FUNCTION_BLOCK SecondState IMPLEMENTS Istate
VAR
	stateFinished: BOOL;
	_description: STRING := 'SecondState';
END_VAR

PROPERTY Description : STRING
GET
END_GET
END_PROPERTY

METHOD execute : BOOL
IF NOT stateFinished THEN 
	THIS^();
END_IF

execute:= stateFinished;
END_METHOD

///FB_Init is always available implicitly and it is used primarily for initialization.
///The return value is not evaluated. For a specific influence, you can also declare the
///methods explicitly and provide additional code there with the standard initialization
///code. You can evaluate the return value.
METHOD FB_Init : BOOL
VAR_INPUT
	/// TRUE: the retain variables are initialized (reset warm / reset cold)
	bInitRetains: BOOL;
	/// TRUE: the instance will be copied to the copy code afterward (online change) 
	bInCopyCode: BOOL;
END_VAR
END_METHOD

END_FUNCTION_BLOCK

(* stored: Version 1.1.0.1
   POU SecondState: Id {efa1cfc3-75fc-4e25-b823-086e67930745}, SpecialFunc None
   Property Description: Id {01ddd6a0-cf9a-4907-841b-9f69f750c812}
   Get Get: Id {557ee3ca-cfc2-47a6-accc-45ec5e733b08}
   Method execute: Id {f2be1b42-2461-459e-b05a-b7ec57fc4abe}
   Method FB_Init: Id {92c893e4-14bd-4bf3-8232-74d76a49a92a} *)
